PROGRAM PRG_ControlSerialLine
VAR
	fbSerialLineControl: SerialLineControl;
	stComInData AT %I*: PcComInData;
	stComOutData AT %Q*: PcComOutData;
END_VAR

fbSerialLineControl(
	Mode:= ComSerialLineMode_t.SERIALLINEMODE_PC_COM_PORT, 
	pComIn:= ADR(stComInData), 
	pComOut:= ADR(stComOutData), 
	SizeComIn:= UINT_TO_INT(SIZEOF(stComInData)), 
	Error=> , 
	ErrorID=> , 
	TxBuffer:= GVL.TxBuffer, 
	RxBuffer:= GVL.RxBuffer);

END_PROGRAM

(* stored: Version 1.1.0.1, ProductVersion 3.1.4024.11
   POU PRG_ControlSerialLine: Id {7f5be57b-29c0-4f35-bdd1-c005db8dca41}, SpecialFunc None *)
